FUNCTION_BLOCK SequentialLightSwitch

VAR CONSTANT
	MAX_OUTPUTS_PER_LEVEL : INT := GVL.MAX_LIGHT_OUTPUTS_PER_LEVEL;
END_VAR

VAR_INPUT
	ID : INT;
	name : STRING := 'Light switch';
	digitalInput : REFERENCE TO BOOL;
	
	small_outputs : REFERENCE TO ARRAY[1..MAX_OUTPUTS_PER_LEVEL] OF BOOL;
	medium_outputs : REFERENCE TO ARRAY[1..MAX_OUTPUTS_PER_LEVEL] OF BOOL;
	big_outputs : REFERENCE TO ARRAY[1..MAX_OUTPUTS_PER_LEVEL] OF BOOL;
	superstrong_outputs : REFERENCE TO ARRAY[1..MAX_OUTPUTS_PER_LEVEL] OF BOOL;
	
	levelsManaged : INT := 3; //max 4
	
	defaultDayOutput : E_OutputLevel;
	defaultNightOutput : E_OutputLevel;
END_VAR

VAR	
	initialized : BOOL := FALSE;
	isOn : BOOL := FALSE;
	smallOutputsSet : BOOL := FALSE;
	mediumOutputsSet : BOOL := FALSE;
	bigOutputsSet: BOOL := FALSE;
	superStrongOutputsSet: BOOL := FALSE;
	
	wasRecentlyActive : BOOL := FALSE;
	pressed : R_TRIG;
	released : F_TRIG;
	smallOutputTimer : TON := (PT := T#1S);
	mediumOutputTimer : TON := (PT := T#2S); 
	bigOutputTimer : TON := (PT := T#3S); 
	superStrongOutputTimer : TON := (PT := T#4S);
	inactivityTimeout : TP := (PT := T#1100MS);
	pressedTimer : TON := (PT := T#10S);
	pressedTimeMiliseconds : INT := 0;
	firstLongPress : BOOL := FALSE;
	turnedOnLongSelector : BOOL := FALSE;
	
	consecutiveClicks : INT := 0;
END_VAR

IF NOT initialized THEN
	initialized := TRUE;	
END_IF

METHOD doSpecialAction : BOOL
VAR_INPUT
END_VAR

VAR
	i: INT;
	groupController : GroupController;
END_VAR
CASE ID OF
		//TODO pamietac
	12:
		GVL.EventLogger.print3(level:=TcEventSeverity.Info, str1:='Special action for button 1 - ', str2:='turning off all lights', str3:=getSource());
		MAIN.groupController.requestLightsOff();
		
	17:
		GVL.EventLogger.print3(level:=TcEventSeverity.Info, str1:='Special action for button 2 - ', str2:='turning on all lights', str3:=getSource());
		MAIN.groupController.requestLightsOnDefault();
		
//	3:
//		GVL.EventLogger.print3(level:=TcEventSeverity.Info, str1:='Special action for button 3 - ', str2:='closing all shutters', str3:=getSource());
//		MAIN.groupController.requestShuttersClose();
		
END_CASE
END_METHOD

METHOD PRIVATE getSource : STRING(255)
VAR_INPUT
END_VAR

VAR
	details : STRING(255);
END_VAR
details := CONCAT(STR1:=' - light switch, ID: ', STR2:=TO_STRING(ID));
details := CONCAT(STR1:=details, STR2:=', digital input: ');
details := CONCAT(STR1:=details, STR2:=TO_STRING(digitalInput));
details := CONCAT(STR1:=details, STR2:=', name: ');
details := CONCAT(STR1:=details, STR2:=name);

getSource := details;
END_METHOD

METHOD PRIVATE inputsOutputsLoop
VAR_INPUT
END_VAR
pressed(CLK:= digitalInput);
released(CLK:= digitalInput);
smallOutputTimer(IN := digitalInput);
mediumOutputTimer(IN := digitalInput);
bigOutputTimer(IN := digitalInput);
superStrongOutputTimer(IN := digitalInput);
inactivityTimeout(IN := digitalInput);
pressedTimer(IN := digitalInput);
turnedOnLongSelector := isTurnedOnLongSelector();
END_METHOD

METHOD PRIVATE isTurnedOnLongSelector : BOOL
VAR_INPUT
END_VAR
isTurnedOnLongSelector := smallOutputsSet OR mediumOutputsSet OR bigOutputsSet OR superStrongOutputsSet;
END_METHOD

METHOD loop
VAR_INPUT
END_VAR

VAR
	number : DINT;
	boool : BOOL;
	str3: INT;
END_VAR
verifyIsTurnedOn();
inputsOutputsLoop();


IF NOT inactivityTimeout.Q THEN
	firstLongPress := FALSE;	
END_IF

IF digitalInput THEN
	IF TIME_TO_INT(pressedTimer.ET) <> 0 THEN
		pressedTimeMiliseconds := TIME_TO_INT(pressedTimer.ET);
	END_IF
END_IF

IF wasRecentlyActive AND NOT digitalInput AND NOT inactivityTimeout.Q THEN	
	GVL.EventLogger.print3(level:= TcEventSeverity.Verbose, str1:='Activity timeout', str2:= '', str3:=getSource());
	consecutiveClicks := 0;
	wasRecentlyActive := FALSE;
END_IF

IF pressed.Q THEN
	GVL.EventLogger.print3(level:=TcEventSeverity.Info, str1:='Button pressed', str2:= '', str3:=getSource());
	consecutiveClicks := consecutiveClicks + 1;
	GVL.EventLogger.print3(level:=TcEventSeverity.Verbose, str1:='consecutiveClicks=', str2:= TO_STRING(consecutiveClicks), str3:=getSource());
	GVL.EventLogger.print3(level:=TcEventSeverity.Verbose, str1:='isOn=', str2:= TO_STRING(isOn), str3:=getSource());
	GVL.EventLogger.print3(level:=TcEventSeverity.Verbose, str1:='firstLongPress=', str2:= TO_STRING(firstLongPress), str3:=getSource());
	
END_IF

IF released.Q THEN
	GVL.EventLogger.print3(level:=TcEventSeverity.Info, str1:='Released after ', str2:= TO_STRING(pressedTimeMiliseconds), str3:=getSource());
	GVL.EventLogger.print3(level:=TcEventSeverity.Verbose, str1:='isOn=', str2:= TO_STRING(isOn), str3:=getSource());
	GVL.EventLogger.print3(level:=TcEventSeverity.Verbose, str1:='turnedOnLongSelector=', str2:= TO_STRING(turnedOnLongSelector), str3:=getSource());
	GVL.EventLogger.print3(level:=TcEventSeverity.Verbose, str1:='firstLongPress=', str2:= TO_STRING(firstLongPress), str3:=getSource());	
	IF isON AND NOT turnedOnLongSelector AND NOT firstLongPress THEN
		GVL.EventLogger.print3(level:=TcEventSeverity.Info, str1:='Lights turned off', str2:= '', str3:=getSource());
		turnOff();
	ELSE		
		GVL.EventLogger.print3(level:=TcEventSeverity.Verbose, str1:='wasRecentlyActive=', str2:= TO_STRING(wasRecentlyActive), str3:=getSource());
		IF pressedTimeMiliseconds >= 0 AND pressedTimeMiliseconds <= 300  THEN
			GVL.EventLogger.print3(level:=TcEventSeverity.Verbose, str1:='Quick press released after ', str2:= TO_STRING(pressedTimeMiliseconds), str3:=getSource());
			GVL.EventLogger.print3(level:=TcEventSeverity.Verbose, str1:='firstLongPress=', str2:= TO_STRING(firstLongPress), str3:=getSource());
			IF NOT firstLongPress THEN
				turnOnDefault();
			END_IF
		ELSE 
			IF pressedTimeMiliseconds > 300 AND pressedTimeMiliseconds < 1000 THEN
				GVL.EventLogger.print3(level:=TcEventSeverity.Verbose, str1:='Long press released after ', str2:= TO_STRING(pressedTimeMiliseconds), str3:=getSource());
				GVL.EventLogger.print3(level:=TcEventSeverity.Verbose, str1:='Turn ON strongest as long press', str2:= '', str3:=getSource());
				turnOnStrongestOutput();
			END_IF 
		END_IF
	END_IF
	
	wasRecentlyActive := TRUE;
	pressedTimeMiliseconds := TIME_TO_INT(pressedTimer.ET);
END_IF

IF consecutiveClicks >= 3 THEN
	consecutiveClicks := 0;
	doSpecialAction();
END_IF

manageLongPress();
END_METHOD

METHOD PRIVATE manageLongPress
VAR_INPUT
END_VAR
IF levelsManaged >= 1 AND TIME_TO_DWORD(pressedTimer.ET) >= 1000 THEN
	IF NOT smallOutputsSet THEN
		setOutputs(outputLevel := E_OutputLevel.SMALL, state := TRUE);
		GVL.EventLogger.print3(level:=TcEventSeverity.Verbose, str1:='Long press turn on output ', str2:=TO_STRING(E_OutputLevel.SMALL), str3:=getSource());
	END_IF
END_IF

IF levelsManaged >= 2 AND TIME_TO_DWORD(pressedTimer.ET) >= 2000 THEN
	IF NOT mediumOutputsSet THEN
		setOutputs(outputLevel := E_OutputLevel.MEDIUM, state := TRUE);
		GVL.EventLogger.print3(level:=TcEventSeverity.Verbose, str1:='Long press turn on output', str2:=TO_STRING(E_OutputLevel.SMALL), str3:=getSource());
	END_IF
END_IF

IF levelsManaged >= 3 AND TIME_TO_DWORD(pressedTimer.ET) >= 3000 THEN
	IF NOT bigOutputsSet THEN
		setOutputs(outputLevel := E_OutputLevel.BIG, state := TRUE);
		GVL.EventLogger.print3(level:=TcEventSeverity.Verbose, str1:='Long press turn on output', str2:=TO_STRING(E_OutputLevel.SMALL), str3:=getSource());
	END_IF
END_IF

IF levelsManaged >= 4 AND TIME_TO_DWORD(pressedTimer.ET) >= 4000 THEN
	IF NOT superStrongOutputsSet THEN
		setOutputs(outputLevel := E_OutputLevel.SUPERSTRONG, state := TRUE);
		GVL.EventLogger.print3(level:=TcEventSeverity.Verbose, str1:='Long press turn on output', str2:=TO_STRING(E_OutputLevel.SMALL), str3:=getSource());
	END_IF
END_IF
END_METHOD

METHOD PRIVATE setOutputs
VAR_INPUT
	outputLevel : E_OutputLevel;
	state : BOOL;
END_VAR

VAR
	i : INT;
	state_as_text : STRING := 'abc';
END_VAR
state_as_text := TO_STRING(state);

CASE outputLevel OF
	
	E_OutputLevel.SMALL:
		GVL.EventLogger.print3(level:=TcEventSeverity.Info, str1:='Set SMALL outputs to: ', str2:= state_as_text, str3:=getSource());
		FOR i := 1 TO MAX_OUTPUTS_PER_LEVEL BY 1 DO
			small_outputs[i] := state;
		END_FOR
		
	E_OutputLevel.MEDIUM:
		GVL.EventLogger.print3(level:=TcEventSeverity.Info, str1:='Set MEDIUM outputs to: ', str2:= state_as_text, str3:=getSource());	
		FOR i := 1 TO MAX_OUTPUTS_PER_LEVEL BY 1 DO
			medium_outputs[i] := state;
		END_FOR
		
	E_OutputLevel.BIG:
		GVL.EventLogger.print3(level:=TcEventSeverity.Info, str1:='Set BIG outputs to: ', str2:= state_as_text, str3:=getSource());
		FOR i := 1 TO MAX_OUTPUTS_PER_LEVEL BY 1 DO
			big_outputs[i] := state;
		END_FOR
		
	E_OutputLevel.SUPERSTRONG:
		GVL.EventLogger.print3(level:=TcEventSeverity.Info, str1:='Set SUPERSTRONG outputs to: ', str2:= state_as_text, str3:=getSource());
		FOR i := 1 TO MAX_OUTPUTS_PER_LEVEL BY 1 DO
			superstrong_outputs[i] := state;
		END_FOR
		
END_CASE
END_METHOD

METHOD PUBLIC turnOff
VAR_INPUT
END_VAR

VAR 
	i : INT;
END_VAR
CASE levelsManaged OF
	1 :
		FOR i := 1 TO MAX_OUTPUTS_PER_LEVEL BY 1 DO
			small_outputs[i] := FALSE;
		END_FOR

	2 :
		FOR i := 1 TO MAX_OUTPUTS_PER_LEVEL BY 1 DO
			small_outputs[i] := FALSE;
			medium_outputs[i] := FALSE;
		END_FOR
	
	3 :
		FOR i := 1 TO MAX_OUTPUTS_PER_LEVEL BY 1 DO
			small_outputs[i] := FALSE;
			medium_outputs[i] := FALSE;
			big_outputs[i] := FALSE;
		END_FOR
		
	4 :
		FOR i := 1 TO MAX_OUTPUTS_PER_LEVEL BY 1 DO
			small_outputs[i] := FALSE;
			medium_outputs[i] := FALSE;
			big_outputs[i] := FALSE;
			superstrong_outputs[i] := FALSE;
		END_FOR

END_CASE

isOn := FALSE;
END_METHOD

METHOD PUBLIC turnOnDefault
VAR_INPUT
END_VAR
IF MAIN.isDay THEN
	GVL.EventLogger.print3(level:=TcEventSeverity.Verbose, str1:='turn ON default for daytime: ', str2:= TO_STRING(defaultDayOutput), str3:=getSource());
	setOutputs(outputLevel := defaultDayOutput, state := TRUE);
ELSE
	GVL.EventLogger.print3(level:=TcEventSeverity.Verbose, str1:='turn ON default for nighttime: ', str2:= TO_STRING(defaultNightOutput), str3:=getSource());
	setOutputs(outputLevel := defaultNightOutput, state := TRUE);
END_IF

isOn := TRUE;
END_METHOD

METHOD turnOnStrongestOutput
VAR_INPUT
END_VAR

VAR
	i : INT;
END_VAR
CASE levelsManaged OF
	1:
		setOutputs(outputLevel := E_OutputLevel.SMALL, state := TRUE);
		setOutputs(outputLevel := E_OutputLevel.MEDIUM, state := FALSE);
		setOutputs(outputLevel := E_OutputLevel.BIG, state := FALSE);
		setOutputs(outputLevel := E_OutputLevel.SUPERSTRONG, state := FALSE);
	2:
		setOutputs(outputLevel := E_OutputLevel.SMALL, state := FALSE);
		setOutputs(outputLevel := E_OutputLevel.MEDIUM, state := TRUE);
		setOutputs(outputLevel := E_OutputLevel.BIG, state := FALSE);
		setOutputs(outputLevel := E_OutputLevel.SUPERSTRONG, state := FALSE);
		
	3:
		setOutputs(outputLevel := E_OutputLevel.SMALL, state := FALSE);
		setOutputs(outputLevel := E_OutputLevel.MEDIUM, state := FALSE);
		setOutputs(outputLevel := E_OutputLevel.BIG, state := TRUE);
		setOutputs(outputLevel := E_OutputLevel.SUPERSTRONG, state := FALSE);
		
	4:
		setOutputs(outputLevel := E_OutputLevel.SMALL, state := FALSE);
		setOutputs(outputLevel := E_OutputLevel.MEDIUM, state := FALSE);
		setOutputs(outputLevel := E_OutputLevel.BIG, state := FALSE);
		setOutputs(outputLevel := E_OutputLevel.SUPERSTRONG, state := TRUE);
		
END_CASE

isOn := TRUE;
END_METHOD

METHOD PRIVATE verifyIsTurnedOn
VAR_INPUT
END_VAR

VAR
	i : INT;
END_VAR
isOn := FALSE;
smallOutputsSet := FALSE;
mediumOutputsSet := FALSE;
bigOutputsSet := FALSE;
superStrongOutputsSet := FALSE;

IF levelsManaged >= 1 THEN
	FOR i := 1 TO MAX_OUTPUTS_PER_LEVEL BY 1 DO
		IF small_outputs[i] = TRUE THEN
			isOn := TRUE;
			smallOutputsSet := TRUE;
		END_IF
	END_FOR
END_IF

IF levelsManaged >= 2 THEN
	FOR i := 1 TO MAX_OUTPUTS_PER_LEVEL BY 1 DO
		IF medium_outputs[i] = TRUE THEN
			isOn := TRUE;
			mediumOutputsSet := TRUE;
		END_IF
	END_FOR
END_IF

IF levelsManaged >= 3 THEN
	FOR i := 1 TO MAX_OUTPUTS_PER_LEVEL BY 1 DO
		IF big_outputs[i] = TRUE THEN
			isOn := TRUE;
			bigOutputsSet := TRUE;
		END_IF
	END_FOR
END_IF

IF levelsManaged >= 4 THEN
	FOR i := 1 TO MAX_OUTPUTS_PER_LEVEL BY 1 DO
		IF superstrong_outputs[i] = TRUE THEN
			isOn := TRUE;
			superStrongOutputsSet := TRUE;
		END_IF
	END_FOR
END_IF


RETURN;
END_METHOD

END_FUNCTION_BLOCK

(* stored: Version 1.1.0.1, ProductVersion 3.1.4024.12
   POU SequentialLightSwitch: Id {aec94d50-ff8e-4733-83a7-9ffb2f475799}, SpecialFunc None
   Method doSpecialAction: Id {6e16f68b-e074-467f-9286-070fb5400126}
   Method getSource: Id {aef894df-032e-4098-aeaf-85b387f704db}
   Method inputsOutputsLoop: Id {e8351a60-1cd2-41ed-9032-90cf759bb181}
   Method isTurnedOnLongSelector: Id {7bae46af-3a44-48ea-bbd6-f40ab3340ff2}
   Method loop: Id {8ef97f03-9ee7-4fed-a21d-d7d2049ac2bc}
   Method manageLongPress: Id {9f04a0be-cdbd-4dba-be58-f2a3e3154f07}
   Method setOutputs: Id {98f0d494-d3da-4ed5-b4b3-67a830019a2c}
   Method turnOff: Id {6af44e6f-dbfa-4c03-a237-33da5be5a32c}
   Method turnOnDefault: Id {0b29667d-d1f0-4d16-a335-62900f4a810a}
   Method turnOnStrongestOutput: Id {3f4fabbe-4d13-4779-9909-6746b7be7f4d}
   Method verifyIsTurnedOn: Id {4e977ce7-4f11-4414-adce-fc6f7d22aa32} *)
